# EPICS autosave request: quadEMApp/Db/quadEM_TimeSeries_settings.req
# FILE... quadEM_TimeSeries_settings.req
$(P)$(R)ReadAll.SCAN
$(P)$(R)NuseAll
$(P)$(R)Dwell
$(P)$(R)PresetReal
$(P)$(R)EnableClientWait
